(* CoDeSys 2.3 export: PV_ST.EXP *)

(* Data type *)
TYPE PV_ST :
	(
	PV_ERROR := 0,
	PV_ISOLATING,
	PV_ISOLATED,
	PV_SLOW_VENTING,
	PV_FAST_VENTING,
	PV_VENTED,
	PV_RP_STARTING,
	PV_RP_PUMPING,
	PV_RP_PUMPED,
	PV_TP_PUMPING,
	PV_PUMPED
	);
END_TYPE
